(* PLC project  *)

CONFIGURATION PLC
END_CONFIGURATION
